{attribute 'pack_mode' := '1'}
TYPE ST_ReadPathData :
STRUCT
	stReadListReturnInfo		: ARRAY [1..1] OF ST_UAReadListReturnInfo;
	stPathData					: ST_StatusPath;

END_STRUCT
END_TYPE

(* stored: Version 1.1.0.1, ProductVersion 3.1.4024.5
   DUT ST_ReadPathData: Id {93ac093b-99fd-4cc9-ba60-73affc2223a2} *)
